Staubli VAL3: reveMarkItem.pgx

public program reveMarkItem(string x_sName)
  local num i
begin
  for i=0 to size(sml:box[x_sName].comment)-1
    if left(sml:box[x_sName].comment[i],1)!="#"
      sml:box[x_sName].comment[i]="# "+sml:box[x_sName].comment[i]
    else
     sml:box[x_sName].comment[i]=right(sml:box[x_sName].comment[i],len(sml:box[x_sName].comment[i])-2)
    endIf
  endFor
end
